SUBAPPLICATION RedGreenBackground4SC (* Hintergrundfarbe (TRUE -> Rot, FALSE -> Grün) für 3 Objekte (Kompakt) *)
  (* Standard: 61499-2 *)
  (* Version 1.0, 2024-01-01, franz *)
  PACKAGE MyLib::sys;
  IMPORT isobus::UT::Q::const::IDs::ID_NULL;
  IMPORT isobus::UT::Q::types::s3ObjectIDs;
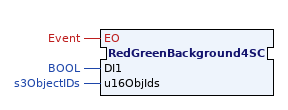
  EVENT_INPUT
    EO;
  END_EVENT
  VAR_INPUT
    DI1 : BOOL; (* Selector *)
    u16ObjIds : isobus::UT::Q::types::s3ObjectIDs := (u16ObjId := ID_NULL, u16ObjIdA := ID_NULL, u16ObjIdB := ID_NULL); (* Object IDs *)
  END_VAR
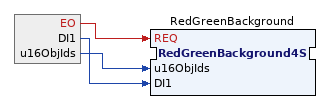
  SUBAPPS
    RedGreenBackground : MyLib::sys::RedGreenBackground4S;
  END_SUBAPPS
  EVENT_CONNECTIONS
    EO TO RedGreenBackground.REQ;
  END_CONNECTIONS
  DATA_CONNECTIONS
    u16ObjIds TO RedGreenBackground.u16ObjIds;
    DI1 TO RedGreenBackground.DI1;
  END_CONNECTIONS
END_SUBAPPLICATION
